FUNCTION_BLOCK FB_Chamber1Endpoint1DoorOpenService EXTENDS FB_ServiceBase
VAR_IN_OUT
	IsDoorClose : BOOL;
	DoorCloseCtrl : BOOL;
END_VAR

M_UpdateService(CompletionBehavior := E_ServiceCompletionBehavior.NaturalCompletion);

METHOD PROTECTED H_OnExecute : E_PackMLHookResult
VAR_INPUT
	bFirstScan : BOOL;
END_VAR
H_OnExecute := E_PackMLHookResult.Busy;

DoorCloseCtrl := FALSE;

IF IsDoorClose = FALSE THEN
	H_OnExecute := E_PackMLHookResult.Done;
END_IF
END_METHOD

END_FUNCTION_BLOCK

(* stored: Version 1.1.0.1, ProductVersion 3.1.4026.18
   POU FB_Chamber1Endpoint1DoorOpenService: Id {4daeed7c-3826-41bd-bf92-bfd659122874}, SpecialFunc None
   Folder StateAction: Id {646b83f4-0787-498b-af58-9cda5139b54e}
   Method H_OnExecute: Id {bf4ab31f-7e62-4525-8a41-8b0a1f44ff39} *)
